FUNCTION_BLOCK FB_Route12to6
VAR
	nStatus		:INT	:=0;
	GreenRight	:FB_GreenConveyor;				//Right Green Conveyor
	GreenLeft	:FB_GreenConveyor;				//Left Green Conveyor
	OrangeUpper	:FB_OrangeConveyor;				//Upper Orange Conveyor
	OrangeLower	:FB_OrangeConveyor;				//Lower Orange Conveyor
END_VAR

CASE nStatus OF
0:	GreenRight.Motor.RunMotor();
	//Reader();
	IF Random.number=6 THEN
	nStatus:=10;
END_IF
10:	IF  GreenRight.LTU.Occupied THEN					//check LTU occupied
		GreenRight.BlueStopper.MoveStopper();			//If occupied move stopper
		ELSE
		GreenRight.LTU.MoveBottom();					//LTU Move bottom to saty on green
		nStatus:=20;									
	END_IF										
20:	IF NOT OrangeLower.LTU.Occupied THEN				//check LTU occupied
				OrangeLower.LTU.MoveBottom();			//LTU Move bottom to saty on green
				nStatus:=30;
				ELSE
				GreenRight.LTU.MoveMiddle();			//LTU Move middle to stop on green
			END_IF
30:	nStatus:=0;
END_CASE

END_FUNCTION_BLOCK

(* stored: Version 1.1.0.1, ProductVersion 3.1.4024.12
   POU FB_Route12to6: Id {3413c003-22a1-4350-96e2-567617198c4a}, SpecialFunc None *)
